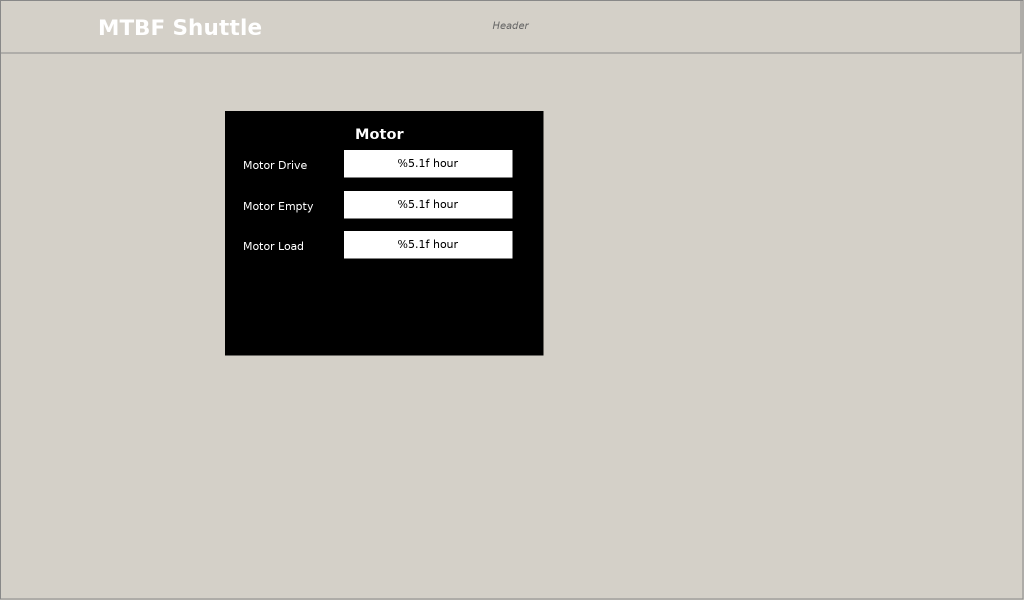
VISUALIZATION MTBF_Shuttle  // 1024x600
    Frame (0,-2 1021x55)
        shows Header()
    Label (95,15 250x25), "MTBF Shuttle"
    RoundedRectangle (225,111 318x244)
    Label (243,114 273x40), "Motor"
    Label (240,148 103x35), "Motor Drive"
    RoundedRectangle (343,149 170x29), "%5.1f hour", text variable: InputOutput_GVL.MTBF_Motor[16]
    Label (240,189 103x35), "Motor Empty"
    RoundedRectangle (343,190 170x29), "%5.1f hour", text variable: InputOutput_GVL.MTBF_Motor[17]
    Label (240,229 103x35), "Motor Load"
    RoundedRectangle (343,230 170x29), "%5.1f hour", text variable: InputOutput_GVL.MTBF_Motor[18]
END_VISUALIZATION

(* stored: Version 1.1.0.1, ProductVersion 3.1.4024.12
   Visu MTBF_Shuttle: Id {b749bd8f-651a-4c4b-8f50-13b5941dbbf1} *)
